PROGRAM MAIN
VAR
END_VAR

TC3PingEsp();

END_PROGRAM

(* stored: Version 1.1.0.1, ProductVersion 3.1.4024.12
   POU MAIN: Id {0e184861-7704-467f-8cc6-a538c89b8fb5}, SpecialFunc None *)
